PROGRAM TactTime
VAR

	TactTime: TactTimeFB;

END_VAR

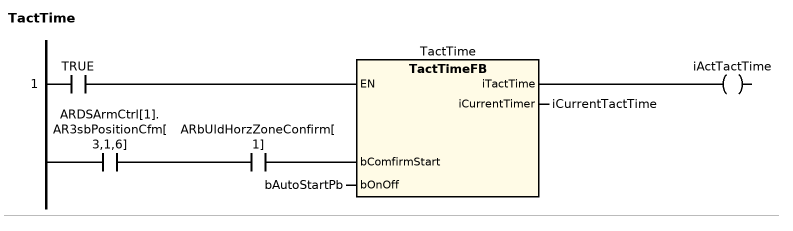
// NETWORK 1
TactTime(
    bComfirmStart := ARDSArmCtrl[1].AR3sbPositionCfm[3,1,6] AND ARbUldHorzZoneConfirm[1],
    bOnOff := bAutoStartPb,
    iCurrentTimer => iCurrentTactTime); // TactTimeFB
iActTactTime := TactTime.iTactTime;

END_PROGRAM

(* stored: Version 1.1.0.1, ProductVersion 3.1.4024.12
   POU TactTime: Id {0ba15a1a-3b2e-48b9-bee9-8c4511b5f644}, SpecialFunc None *)
